FUNCTION_BLOCK carousel_belt
  (* Standard: 61499-2 *)
  (* Version 0,1, 2015-00-16, Th?o, PC_THEO *)
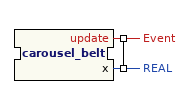
  EVENT_OUTPUT
    update WITH x;
  END_EVENT
  VAR_OUTPUT
    x : REAL;
  END_VAR
  VAR
    beta : REAL;
  END_VAR
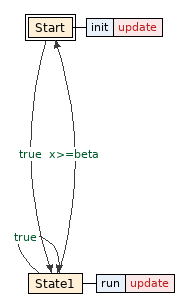
  EC_STATES
    Start : init -> update;
    State1 : run -> update;
  END_STATES
  EC_TRANSITIONS
    Start TO State1 := true;
    State1 TO Start := x>=beta;
    State1 TO State1 := true;
  END_TRANSITIONS
  ALGORITHM init IN C:
me->x=0;
me->beta=10;
  END_ALGORITHM
  ALGORITHM run IN C:
me->x=me->x+1;
//printf("icecream, %f\n", me->x);
  END_ALGORITHM
END_FUNCTION_BLOCK
